PROGRAM P_Betriebsarten
VAR
	
END_VAR

(* Baustein: FC2 - Start,Stop,Betriebsarten *)
(* FC2 - AWL2ST: Fertig *)

F_EndschalterBruecken(); // OK 

P_FlankenErzeugen(); // OK 

P_BlinktaktTastleuchten(); // OK

F_StartStopTipp(); // OK

END_PROGRAM

(* stored: Version 1.1.0.1, ProductVersion 3.1.4024.3
   POU P_Betriebsarten: Id {e5518de6-ec41-4738-9477-6ecda80f2f0d}, SpecialFunc None *)
